(* CoDeSys 2.3 export: FB_FCModbusInterface.exp *)

(* POU 02_DeviceControl/FrequencyConverter/VAR_INPUT, ST *)
FUNCTION_BLOCK

VAR_INPUT
    stModbusData: ST_FC_ModbusData;    (* ґРЭЭлХ Юв Modbus *)
    xModbusOK: BOOL;                   (* єРзХбвТЮ бТпЧШ *)   
END_VAR

VAR_OUTPUT
    stStatus: ST_FC_Status;            (* ґХЪЮФШаЮТРЭЭлЩ бвРвгб *)
    stProcessData: ST_FC_ProcessData;  (* ѕСаРСЮвРЭЭлХ ФРЭЭлХ ЯаЮжХббР *)
END_VAR


END_FUNCTION_BLOCK

END_FUNCTION_BLOCK
